// TIA Portal V19 export
FUNCTION_BLOCK "TYPIC_C106_IF_REL"   // FB81, FBD
TITLE = TYPIC_C106_IF_REL: Beveilingsrelais
{ S7_Optimized_Access := 'TRUE' }
AUTHOR : OCOTECH
FAMILY : Typical
NAME : C106.703
// Logisch Object Besturing: C106.703
// 
// De interne functie Beveiligingsrelais verzorgt de bewaking van een beveiligingsrelais.
// stored: MemoryReserve 10, SetENOAutomatically false
   VAR_INPUT
      EXT_AUT { ExternalAccessible := 'False'; ExternalVisible := 'False'; ExternalWritable := 'False'} : Bool;   // Externe (hoofd) beveiliging (1 = OK)
      EXT_HW { ExternalAccessible := 'False'; ExternalVisible := 'False'; ExternalWritable := 'False'} : Bool;   // Sturings hardware (PLC) bewaking (1 = OK)
      CFG_SYNC { ExternalAccessible := 'False'; ExternalVisible := 'False'; ExternalWritable := 'False'} : Bool;   // Type beveiligingsrelais: TRUE = Lijndifferentieel-beveiligingsrelais FALSE = Overstroom-beveiligingsrelais
      IN_STO_NOK { ExternalAccessible := 'False'; ExternalVisible := 'False'; ExternalWritable := 'False'} : Bool;   // Storing aanwezig die niet observeerbaar tot gevolg heeft
      IN_STO_OK { ExternalAccessible := 'False'; ExternalVisible := 'False'; ExternalWritable := 'False'} : Bool;   // Storing aanwezig die observeerbaarheid niet beinvloed
      IN_REL_ALM { ExternalAccessible := 'False'; ExternalVisible := 'False'; ExternalWritable := 'False'} : Bool;   // Alarm per beveiligingsrelais per uitschakelbevel: TRUE = OK / FALSE = Alarm
      IN_AUT_TOE { ExternalAccessible := 'False'; ExternalVisible := 'False'; ExternalWritable := 'False'} : Bool;   // Vermogenschakelaar TOE (gesloten)
      IN_SCA_TOE { ExternalAccessible := 'False'; ExternalVisible := 'False'; ExternalWritable := 'False'} : Bool;   // Aardingschakelaar TOE (gesloten)
      IN_SYNC { ExternalAccessible := 'False'; ExternalVisible := 'False'; ExternalWritable := 'False'} : Bool;   // Lijndifferentieel beveiligingsrelais loopt synchroon
      IN_AUT_C106 { ExternalAccessible := 'False'; ExternalVisible := 'False'; ExternalWritable := 'False'} : Bool;   // Beveiligingen: serie geschakelde terugmelding (1 = OK)
   END_VAR
   VAR_OUTPUT
      VAR_IF_REL { ExternalAccessible := 'False'; ExternalVisible := 'False'; ExternalWritable := 'False'} : "C106_VAR_IF_REL_TYPIC";   // Struct met alle variabelen naar bovenliggende functies
   END_VAR
   VAR
      STO { ExternalWritable := 'False'} : Struct   // Storingen
         A001 : Bool;   // Beveiliging aangesproken
         A002 : Bool;   // Beveiligingsrelais in storing
         A003 : Bool;   // Algemene storing beveiligingsrelais
         A004 : Bool;   // Alarm beveiligingsrelais: Uitschakelbevel
         A005 : Bool;   // Lijndifferentieel-beveiligingsrelais loopt niet synchroon met zijn tegenhanger
      END_STRUCT;
      VAR { ExternalWritable := 'False'} : Struct   // Variabelen
         ALM { ExternalAccessible := 'False'; ExternalVisible := 'False'} : Bool;   // Alarm per beveiligingsrelais per uitschakelbevel: TRUE = OK / FALSE = Alarm
         AUT_TOE { ExternalAccessible := 'False'; ExternalVisible := 'False'} : Bool;   // Vermogenschakelaar TOE (gesloten)
         SCA_TOE { ExternalAccessible := 'False'; ExternalVisible := 'False'} : Bool;   // Aardingschakelaar TOE (gesloten)
         SYNC { ExternalAccessible := 'False'; ExternalVisible := 'False'} : Bool;   // Lijndifferentieel beveiligingsrelais loopt synchroon
         EXT_AUT { ExternalAccessible := 'False'; ExternalVisible := 'False'} : Bool;   // Externe (hoofd) beveiliging aangesproken
         EXT_HW { ExternalAccessible := 'False'; ExternalVisible := 'False'} : Bool;   // Sturings hardware (PLC) in storing
      END_STRUCT;
   END_VAR
BEGIN

REGION Network 1: START
END_REGION

REGION Network 2: +++ Verwerking meetwaarden en statussen +++
   // De meetwaarde en status wordt ontvangen vanuit de interne sturing.
END_REGION

REGION Network 3: +++ Storingen +++
   // Verwerken van de storingsmeldingen (inputs).
END_REGION

REGION Network 4: Storing A001: Beveiliging aangesproken
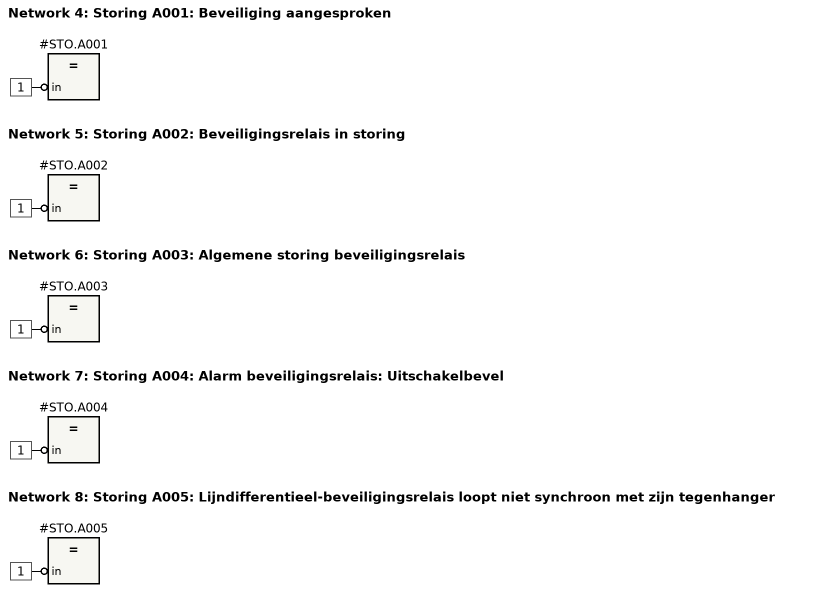
   #STO.A001 := NOT 1;
END_REGION

REGION Network 5: Storing A002: Beveiligingsrelais in storing
   #STO.A002 := NOT 1;
END_REGION

REGION Network 6: Storing A003: Algemene storing beveiligingsrelais
   #STO.A003 := NOT 1;
END_REGION

REGION Network 7: Storing A004: Alarm beveiligingsrelais: Uitschakelbevel
   #STO.A004 := NOT 1;
END_REGION

REGION Network 8: Storing A005: Lijndifferentieel-beveiligingsrelais loopt niet synchroon met zijn tegenhanger
   #STO.A005 := NOT 1;
END_REGION

REGION Network 9 (SCL): EINDE
   // Variabelen van intern scada rakvlak naar outputs copieren
   #VAR_IF_REL.ALM := #VAR.ALM;
   #VAR_IF_REL.AUT_TOE := #VAR.AUT_TOE;
   #VAR_IF_REL.SCA_TOE := #VAR.SCA_TOE;
   #VAR_IF_REL.SYNC := #VAR.SYNC;
   #VAR_IF_REL.EXT_AUT := #VAR.EXT_AUT;
   #VAR_IF_REL.EXT_HW := #VAR.EXT_HW;
END_REGION
END_FUNCTION_BLOCK
